(* Logix 5000 project; controller EIB_Test_PLC vendor 1 type 14 code 107 rev 36.11; software revision 36.00 *)
// External Interface Board Test

TASK MainTask (continuous, watchdog 500 ms) : MainProgram

MODULES
   Local : vendor 1 type 14 code 107 (Compact 0, rev 36.11)
       : vendor 1 type 7 code 66 (Compact 3, rev 2.1, Output RPI 20 ms)
      DO1 : 1769-OB16 (Compact 1, rev 2.1, Output RPI 20 ms)
      DO2 : 1769-OB16 (Compact 2, rev 2.1, Output RPI 20 ms)
END_MODULES

VAR_GLOBAL   (* controller tags *)
   CR0 : BOOL;
   CR1 : BOOL;
   CR2 : BOOL;
   CR3 : BOOL;
   DO1_0 : BOOL;
   DO1_1 : BOOL;
   DO1_10 : BOOL;
   DO1_11 : BOOL;
   DO1_12 : BOOL;
   DO1_13 : BOOL;
   DO1_14 : BOOL;
   DO1_15 : BOOL;
   DO1_2 : BOOL;
   DO1_3 : BOOL;
   DO1_4 : BOOL;
   DO1_5 : BOOL;
   DO1_6 : BOOL;
   DO1_7 : BOOL;
   DO1_8 : BOOL;
   DO1_9 : BOOL;
   DO2_0 : BOOL;
   DO2_1 : BOOL;
   DO2_10 : BOOL;
   DO2_11 : BOOL;
   DO2_12 : BOOL;
   DO2_13 : BOOL;
   DO2_14 : BOOL;
   DO2_15 : BOOL;
   DO2_2 : BOOL;
   DO2_3 : BOOL;
   DO2_4 : BOOL;
   DO2_5 : BOOL;
   DO2_6 : BOOL;
   DO2_7 : BOOL;
   DO2_8 : BOOL;
   DO2_9 : BOOL;
END_VAR

PROGRAM MainProgram   (* main routine MainRoutine *)

ROUTINE MainRoutine   (* ladder *)
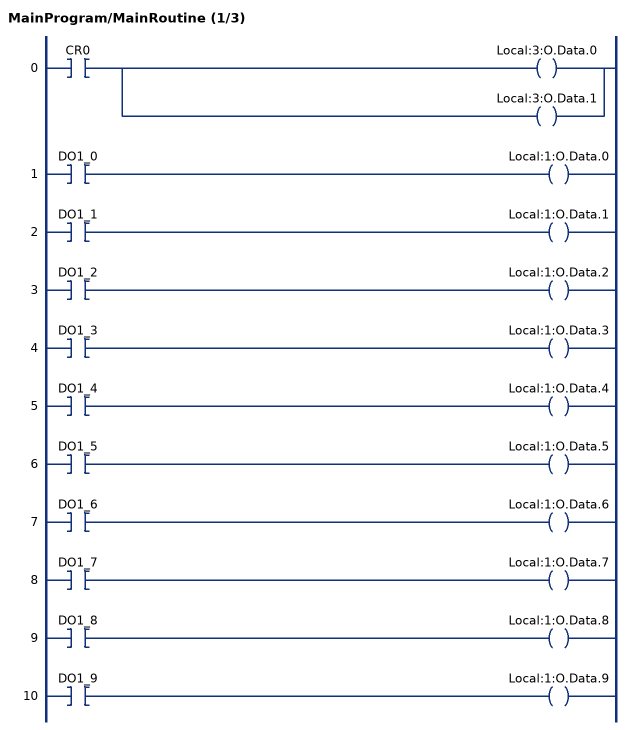
   0: XIC(CR0)[OTE(Local:3:O.Data.0) ,OTE(Local:3:O.Data.1) ];
   1: XIC(DO1_0)OTE(Local:1:O.Data.0);
   2: XIC(DO1_1)OTE(Local:1:O.Data.1);
   3: XIC(DO1_2)OTE(Local:1:O.Data.2);
   4: XIC(DO1_3)OTE(Local:1:O.Data.3);
   5: XIC(DO1_4)OTE(Local:1:O.Data.4);
   6: XIC(DO1_5)OTE(Local:1:O.Data.5);
   7: XIC(DO1_6)OTE(Local:1:O.Data.6);
   8: XIC(DO1_7)OTE(Local:1:O.Data.7);
   9: XIC(DO1_8)OTE(Local:1:O.Data.8);
   10: XIC(DO1_9)OTE(Local:1:O.Data.9);
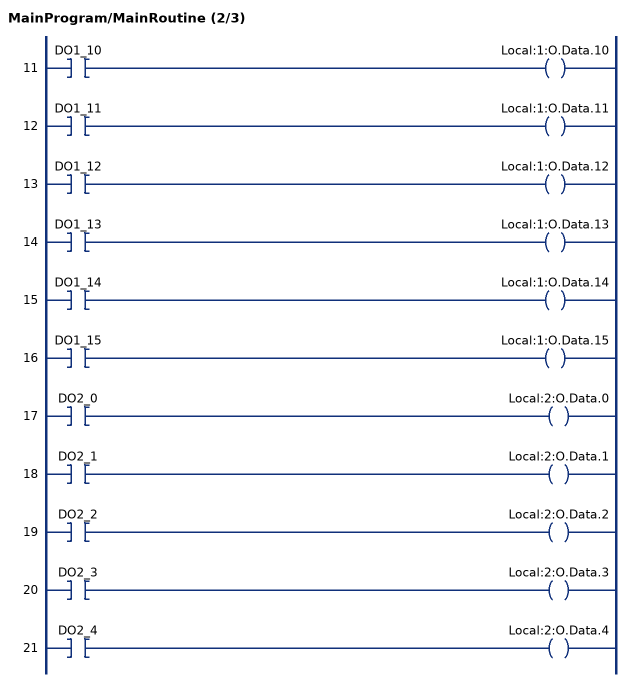
   11: XIC(DO1_10)OTE(Local:1:O.Data.10);
   12: XIC(DO1_11)OTE(Local:1:O.Data.11);
   13: XIC(DO1_12)OTE(Local:1:O.Data.12);
   14: XIC(DO1_13)OTE(Local:1:O.Data.13);
   15: XIC(DO1_14)OTE(Local:1:O.Data.14);
   16: XIC(DO1_15)OTE(Local:1:O.Data.15);
   17: XIC(DO2_0)OTE(Local:2:O.Data.0);
   18: XIC(DO2_1)OTE(Local:2:O.Data.1);
   19: XIC(DO2_2)OTE(Local:2:O.Data.2);
   20: XIC(DO2_3)OTE(Local:2:O.Data.3);
   21: XIC(DO2_4)OTE(Local:2:O.Data.4);
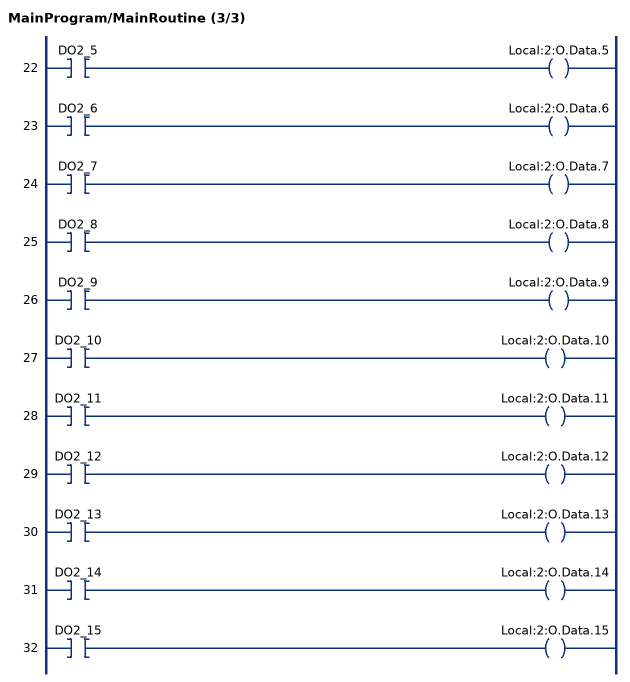
   22: XIC(DO2_5)OTE(Local:2:O.Data.5);
   23: XIC(DO2_6)OTE(Local:2:O.Data.6);
   24: XIC(DO2_7)OTE(Local:2:O.Data.7);
   25: XIC(DO2_8)OTE(Local:2:O.Data.8);
   26: XIC(DO2_9)OTE(Local:2:O.Data.9);
   27: XIC(DO2_10)OTE(Local:2:O.Data.10);
   28: XIC(DO2_11)OTE(Local:2:O.Data.11);
   29: XIC(DO2_12)OTE(Local:2:O.Data.12);
   30: XIC(DO2_13)OTE(Local:2:O.Data.13);
   31: XIC(DO2_14)OTE(Local:2:O.Data.14);
   32: XIC(DO2_15)OTE(Local:2:O.Data.15);
END_ROUTINE
END_PROGRAM
